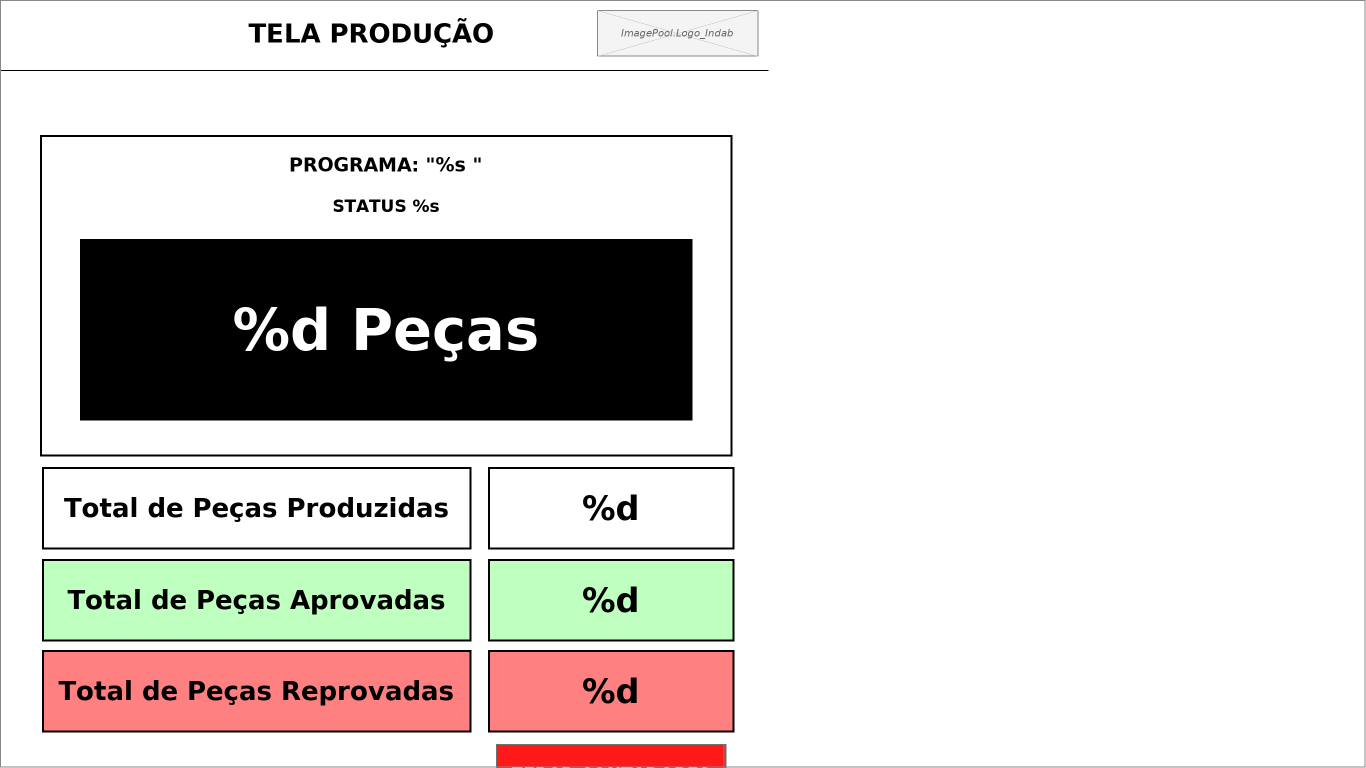
VISUALIZATION Tela_Producao  // 1366x768
    Line (0,1312) (768,1312)
    Rectangle (584,1340 180x24), "%t[dd/MM/yyyy]"
    Rectangle (584,1316 180x24), "%t[HH:mm:ss]"
    Group (0,7 768x64)
        Line (0,63) (768,63)
        Image (597,3 161x46), image: ImagePool.Logo_Indab
        Label (153,0 437x53), "TELA PRODUÇÃO"
    RoundedRectangle (40,135 692x321)
    RoundedRectangle (80,239 612x181), "%d Peças", text variable: Contador_Total
    Rectangle (81,147 610x36), "PROGRAMA: "%s "", text variable: Recipe_name_Select
    RoundedRectangle (42,467 429x82), "Total de Peças Produzidas"
    RoundedRectangle (488,467 246x82), "%d", text variable: Contador_Total
    RoundedRectangle (42,559 429x82), "Total de Peças Aprovadas"
    RoundedRectangle (488,559 246x82), "%d", text variable: Contador_PecasAprovadas
    RoundedRectangle (42,650 429x82), "Total de Peças Reprovadas"
    RoundedRectangle (488,650 246x82), "%d", text variable: Contador_PecasReprovadas
    RoundedRectangle (40,901 692x400)
    Button (496,744 230x60), "ZERAR CONTADORES"
        OnMouseClick: execute { BT_ihm_zerar_contador := TRUE; }
    Rectangle (80,925 610x35), "COMANDOS", text variable: Recipe_name_Select
    Button (15,1315 175x45), "RECEITAS"
        OnMouseClick: change screen: Tela_Receita
    Button (195,1315 175x45), "MANUTENÇÃO"
        OnMouseClick: change screen: Tela_Manutencao
    Rectangle (81,188 610x36), "STATUS %s"
    Button (375,1315 175x45), "ALARMES"
        OnMouseClick: change screen: Tela_Alarmes_1
    PowerSwitch (515,1075 143x136), variable: IhmBt_Desligar, behaviour: TOGGLE, style: Switch-PowerSwitch-Red
    PushSwitch (123,1034 90x90), variable: IhmBt_Ligar, behaviour: TOGGLE, style: Switch-PushSwitch-Green
    Rectangle (115,1000 106x38), "START", text variable: Recipe_name_Select
    PushSwitch (123,1184 90x90), variable: IhmBt_Reset, behaviour: TAP, style: Switch-PushSwitch-Blue
    Rectangle (115,1150 106x38), "RESET", text variable: Recipe_name_Select
    PushSwitch (323,1034 90x90), variable: IhmBt_Pausar, behaviour: TOGGLE, style: Switch-PushSwitch-Yellow
    Rectangle (315,1000 106x38), "PAUSE", text variable: Recipe_name_Select
    Rectangle (538,1031 106x38), "STOP", text variable: Recipe_name_Select
    Rectangle (278,1150 180x38), "COND. INICIAIS", text variable: Recipe_name_Select
    PushSwitch (323,1184 90x90), variable: IhmBt_CondIniciais, behaviour: TOGGLE, style: Switch-PushSwitch-Yellow
    Image (630,900 100x100), invisible if: NOT MaquinaAlarme, image: VisuSymbols.Symbols.Caution
    Button (496,810 230x60), "MODO: %s", text variable: IhmBt_ManualAuto_Text, colour toggle: IhmBt_ManualAuto_Color
        toggle IhmBt_ManualAuto
END_VISUALIZATION

(* stored: Version 1.1.0.1, ProductVersion 3.1.4024.11
   Visu Tela_Producao: Id {7380d848-5c2e-491a-964f-7f324bfb6f4f} *)
